{attribute 'qualified_only'}
{attribute 'strict'}
TYPE E_SaMChangeCategory :
(
	eState		:= 0,
	eMode		:= 1
);
END_TYPE

(* stored: Version 1.1.0.1
   DUT E_SaMChangeCategory: Id {46c4c65d-bc0e-0775-3146-f0582e49e95d} *)
